// TIA Portal V18 export
TYPE "PLCtoMES_ProcessData"
// stored: IsFailsafeCompliant false
   STRUCT
      SubResult : Byte;   // 分项合格状态1 1-合格 2-不合格 3-强制合格
      SubUSL : Real;   // 结果值x规格上限
      SubResultValue : Real;   // 结果值x
      SubLSL : Real;   // 结果值x规格下限
   END_STRUCT;
END_TYPE
